VAR_GLOBAL
	Cell_Pos1 AT %I* : BOOL;
	Cell_Pos2 AT %I* : BOOL;
	Cell_Pos3 AT %I* : BOOL;
	
	Cell_Pos4 AT %I* : BOOL;
	Cell_Pos5 AT %I* : BOOL;
	Cell_Pos6 AT %I* : BOOL;
END_VAR

(* stored: Version 1.1.0.1, ProductVersion 3.1.4026.11
   GVL GVL_CellPositionSensors: Id {324b8032-1e77-45c9-b1c7-509f023d8566} *)
